Staubli VAL3: start.pgx

program start()
begin
  call initdata()
  waitEndMove()
  delay(0)
  taskCreate "RobotMotion",100,RobotMotion()
  taskCreate "CmdTxtReading",85,CmdTxtReading()
  //  taskCreateSync "CmdTxtReading",0.004,btrig,CmdTxtReading()

  taskCreateSync "PositionTrigger",0.01,btrig,PositionTrigger()
end
